% RSLogix 500 project ST_LIGHT_BAK003.RSS, saved by version 8.30.00.16 %
PROJECT "ST_LIGHT"    % processor: Bul.1763 MicroLogix 1100 Series B %

PROGRAM FILES
  LAD 2 "MAIN"  3 rungs
  LAD 3 "LIGHT_SYS"  11 rungs
  LAD 4 "HMI"  1 rungs

DATA FILES
  O0 OUTPUT  4 elements
  I1 INPUT  6 elements
  S2 STATUS  66 elements
  B3 BINARY  1 elements
  T4 TIMER  4 elements
  C5 COUNTER  1 elements
  R6 CONTROL  1 elements
  N7 INTEGER  1 elements
  F8 FLOAT  1 elements

LADDER 2 "MAIN"
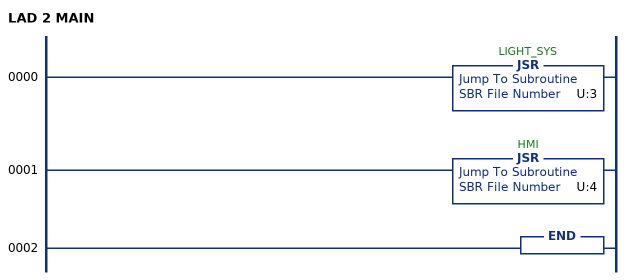
% Rung: 0 %
SOR JSR U:3 EOR
%   U:3  LIGHT_SYS %
% Rung: 1 %
SOR JSR U:4 EOR
%   U:4  HMI %
% Rung: 2 %
SOR END EOR

LADDER 3 "LIGHT_SYS"
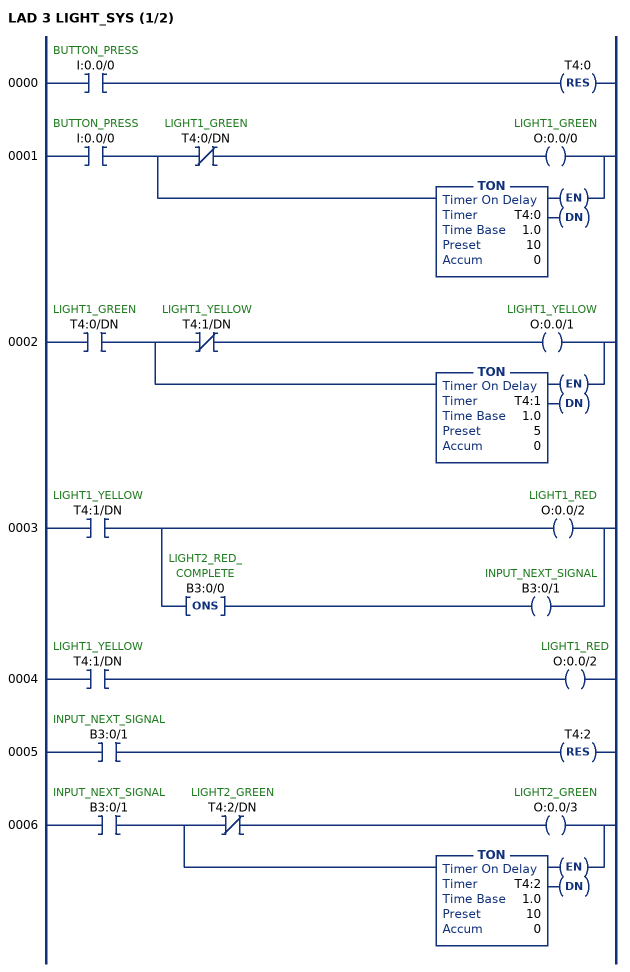
% Rung: 0 %
SOR XIC I:0.0/0 RES T4:0 EOR
%   I:0.0/0  BUTTON_PRESS %
% Rung: 1 %
SOR XIC I:0.0/0 BST XIO T4:0/DN OTE O:0.0/0 NXB TON T4:0 1.0 10 0 BND EOR
%   I:0.0/0  BUTTON_PRESS %
%   T4:0/DN  "LIGHT1_GREEN" %
%   O:0.0/0  LIGHT1_GREEN %
% Rung: 2 %
SOR XIC T4:0/DN BST XIO T4:1/DN OTE O:0.0/1 NXB TON T4:1 1.0 5 0 BND EOR
%   T4:0/DN  "LIGHT1_GREEN" %
%   T4:1/DN  "LIGHT1_YELLOW" %
%   O:0.0/1  LIGHT1_YELLOW %
% Rung: 3 %
SOR XIC T4:1/DN BST OTE O:0.0/2 NXB ONS B3:0/0 OTE B3:0/1 BND EOR
%   T4:1/DN  "LIGHT1_YELLOW" %
%   O:0.0/2  LIGHT1_RED %
%   B3:0/0  LIGHT2_RED_COMPLETE %
%   B3:0/1  INPUT_NEXT_SIGNAL %
% Rung: 4 %
SOR XIC T4:1/DN OTE O:0.0/2 EOR
%   T4:1/DN  "LIGHT1_YELLOW" %
%   O:0.0/2  LIGHT1_RED %
% Rung: 5 %
SOR XIC B3:0/1 RES T4:2 EOR
%   B3:0/1  INPUT_NEXT_SIGNAL %
% Rung: 6 %
SOR XIC B3:0/1 BST XIO T4:2/DN OTE O:0.0/3 NXB TON T4:2 1.0 10 0 BND EOR
%   B3:0/1  INPUT_NEXT_SIGNAL %
%   T4:2/DN  "LIGHT2_GREEN" %
%   O:0.0/3  LIGHT2_GREEN %

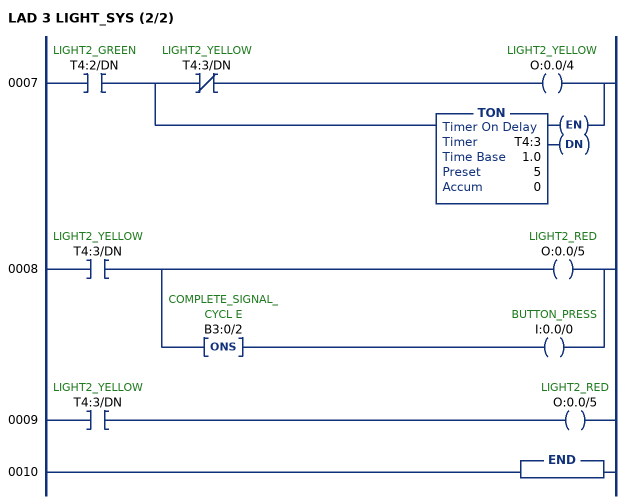
% Rung: 7 %
SOR XIC T4:2/DN BST XIO T4:3/DN OTE O:0.0/4 NXB TON T4:3 1.0 5 0 BND EOR
%   T4:2/DN  "LIGHT2_GREEN" %
%   T4:3/DN  "LIGHT2_YELLOW" %
%   O:0.0/4  LIGHT2_YELLOW %
% Rung: 8 %
SOR XIC T4:3/DN BST OTE O:0.0/5 NXB ONS B3:0/2 OTE I:0.0/0 BND EOR
%   T4:3/DN  "LIGHT2_YELLOW" %
%   O:0.0/5  LIGHT2_RED %
%   B3:0/2  "COMPLETE_SIGNAL_CYCL E" %
%   I:0.0/0  BUTTON_PRESS %
% Rung: 9 %
SOR XIC T4:3/DN OTE O:0.0/5 EOR
%   T4:3/DN  "LIGHT2_YELLOW" %
%   O:0.0/5  LIGHT2_RED %
% Rung: 10 %
SOR END EOR

OTHER DOCUMENTED ADDRESSES
  COMPLETE_CYCLE  
  I:0.0/1  "INPUT TO ANOTHER SIGNAL"
  LIGHT1_COMPLETE_ONS  

DATA TABLE (non-zero values as saved)
DATA T4
% .PRE .ACC %
% T4:0 % 10 0
% T4:1 % 5 0
% T4:2 % 10 0
% T4:3 % 5 0
